{attribute 'qualified_only'}
VAR_GLOBAL
	variable1 : BOOL;
	VarInt: INT;
END_VAR

(* stored: Version 1.1.0.1, ProductVersion 3.1.4024.12
   GVL GVL_1: Id {3b3328bf-e8d6-4166-bc97-3be05e2d34a6} *)
